(* CODESYS project Untitled1.project
   Version: 0.0.0.0
   Title: Untitled1
   Author: madsw

Project tree, tasks and I/O mapping:
  PeackPiercePredatorPendulumProtagonistINATOR_5000 : TM241CEC24T/U, Schneider Electric, order no. TM241CEC24T/U, version 5.0.8.2
      settings: OPCUA enable = True; Dummy int param for online change = 2
    application Application
      libraries: HttpHandling, 1.1.4.0 (Schneider Electric); SysMem, 3.5.12.0 (System); TcpUdpCommunication, 2.0.15.0 (Schneider Electric)
      task MAST (cyclic, interval 300 ms, priority 16, watchdog 100 ms x 1) calls SR_Main
      task MAST_1 (cyclic, interval 100 ms, priority 15, watchdog 50 ms x 1) calls POU
      task Task3 (cyclic, interval 1 ms, priority 1) calls counter
      task VISU_TASK (cyclic, interval 100 ms, priority 31) calls VisuElems.Visu_Prg
      global variables GVL
      program SR_Main [ST]
      POU - Error check functions/
        function CheckBounds [ST]
        function CheckDivDInt [ST]
        function CheckDivLInt [ST]
        function CheckDivReal [ST]
        function CheckDivLReal [ST]
        function CheckPointer [ST]
        function CheckRangeSigned [ST]
        function CheckRangeUnsigned [ST]
        function CheckLRangeSigned [ST]
        function CheckLRangeUnsigned [ST]
      program POU [ST]
      trace Trace (task ): SR_Main.do_Q0
      visualisation Visualization
      program counter [ST]
      OPCUASymbolConfiguration
    DI : Digital Inputs, Schneider Electric, version 5.0.8.2
        settings: IOs Usage = 3
        input  iwDI_IW0 : WORD  // IW0
        input  ibDI_IB1 : BYTE  // IB1
    DQ : Digital Outputs, Schneider Electric, version 5.0.8.2
        output Application.POU.lightArray[0] : BOOL  // QW0.Q0
        output Application.POU.lightArray[1] : BOOL  // QW0.Q1
        output Application.POU.lightArray[2] : BOOL  // QW0.Q2
        output Application.POU.lightArray[3] : BOOL  // QW0.Q3
        output Application.POU.lightArray[4] : BOOL  // QW0.Q4
        output Application.POU.lightArray[5] : BOOL  // QW0.Q5
        output Application.POU.lightArray[6] : BOOL  // QW0.Q6
        output Application.POU.lightArray[7] : BOOL  // QW0.Q7
        output Application.POU.lightArray[8] : BOOL  // QW0.Q8
        output Application.POU.lightArray[9] : BOOL  // QW0.Q9
        output qbDQ_QB1 : BYTE  // QB1
        unmapped channels: QW0
    Counters : Counters, Schneider Electric, version 5.0.8.2
        settings: Instance name = 'HscMainDualPhase_0'; B input History = 'old=-1 new=1'; A input History = 'old=-1 new=0'; Temporary Instance name = 'HscMainDualPhase_0'
    Pulse_Generators : Pulse Generators, Schneider Electric, version 5.0.8.2
    Cartridge_1 : Cartridge, Schneider Electric, version 5.0.8.2
    IO_Bus : IO bus - TM3, Schneider Electric, version 5.0.8.2
      Module_1 : TM3SAF5R/G, Schneider Electric, order no. TM3SAF5R/G, version 1.0.1.14
          input  iwModule_1_IW0 : WORD  // IW0
          output qbModule_1_QB0 : BYTE  // QB0
      Module_2 : TM3AQ4/G, Schneider Electric, order no. TM3AQ4/G, version 1.0.0.15
          output qiModule_2_QW0 : INT  // QW0
          output qiModule_2_QW1 : INT  // QW1
          output qiModule_2_QW2 : INT  // QW2
          output qiModule_2_QW3 : INT  // QW3
          input  ibModule_2_IBStatusQW0 : BYTE  // IBStatusQW0
          input  ibModule_2_IBStatusQW1 : BYTE  // IBStatusQW1
          input  ibModule_2_IBStatusQW2 : BYTE  // IBStatusQW2
          input  ibModule_2_IBStatusQW3 : BYTE  // IBStatusQW3
    COM_Bus : COM bus, Schneider Electric, version 5.0.8.2
    Ethernet_1 : Ethernet Network, Schneider Electric, version 5.0.8.2
        settings: IPAddress = [192, 168, 0, 50]; SubnetMask = [255, 255, 255, 0]; WebServer = TRUE; FTP Server = FALSE; SoMachine Protocol = TRUE; Modbus Server = FALSE; NetManage Protocol = TRUE; SNMP protocol = FALSE; Enable Routing = FALSE; WebVisu protocol = TRUE; DHCP Server Active = TRUE
    Serial_Line_1 : Serial line, Schneider Electric, version 5.0.8.2
      Machine_Expert_Network_Manager : Machine Expert-Network Manager, Schneider Electric, version 4.0.0.3
    Serial_Line_2 : Serial line, Schneider Electric, version 5.0.8.2
      Modbus_Manager : Modbus Manager, Schneider Electric, version 4.0.0.3
    CAN_1 : CANopen bus, Schneider Electric, version 5.0.8.2
  FdtConnections : FDT Connections, Schneider Electric, version 1.0.0.2
  libraries: VisuSymbols, 3.5.10.0 (System)
  CNC settings
  text list GlobalTextList
*)

// PeackPiercePredatorPendulumProtagonistINATOR_5000/Application/GVL
{attribute 'qualified_only'}
VAR_GLOBAL
	gLightArray: ARRAY[0..8] OF BOOL;
	count: UINT;
	
	// OPC UA varibels for interface.
	G_angle: UINT := 45;
END_VAR

// PeackPiercePredatorPendulumProtagonistINATOR_5000/Application/SR_Main
PROGRAM SR_Main
// Comment
VAR
	di_I0: BOOL;
	count: UINT := 4;
	do_Q0: BOOL;
	TCPClient: TCPUDP.FB_TCPClient;
	TCPServer: TCPUDP.FB_TCPServer;
	readBuffer: BYTE;
	PID: PID;
	PD: PD;
END_VAR;

// Global light
GVL.gLightArray[count] := FALSE;
IF count >= 8 THEN
	count := 0;
ELSE
	count := count +1;	
END_IF;
GVL.gLightArray[count] := TRUE;

do_Q0 := NOT NOT NOT di_I0;


HscMainDualPhase_0.CurrentValue;
// TCPClient.Receive(ADR(readBuffer), SIZEOF(BYTE), );

END_PROGRAM

// PeackPiercePredatorPendulumProtagonistINATOR_5000/Application/POU
PROGRAM POU
VAR
	lightArray: ARRAY[0..9] OF BOOL;
	count: UINT;
END_VAR

lightArray[count] := FALSE;
GVL.gLightArray[count] := FALSE;

IF count+1 = SIZEOF(lightArray)/SIZEOF(BOOL) THEN
	count := 0;
ELSE
	count := count +1;	
END_IF;

lightArray[count] := TRUE;
GVL.gLightArray[count] := TRUE;

END_PROGRAM

// PeackPiercePredatorPendulumProtagonistINATOR_5000/Application/counter
PROGRAM counter
VAR
	ctu: CTUD;
	adasd: CTUD;
END_VAR

END_PROGRAM

// PeackPiercePredatorPendulumProtagonistINATOR_5000/Application/POU - Error check functions/CheckBounds
// Implicitly generated code : DO NOT EDIT
FUNCTION CheckBounds : DINT
VAR_INPUT
	index, lower, upper: DINT;
END_VAR

// Implicitly generated code : Only an Implementation suggestion
IF  index < lower THEN
	CheckBounds := lower;
ELSIF  index > upper THEN
	CheckBounds := upper;
ELSE  
	CheckBounds := index;
END_IF

(*It is also possible to set a breakpoint, log messages or e.g. to halt on an exception:
Add CmpApp.library, SysExcept.library and SysTypes2_Itf as newest.
Declaration:
VAR
    _pApp : POINTER TO CmpApp.APPLICATION;
    _result   : SysTypes.RTS_IEC_RESULT;
END_VAR

Implementation:
_pApp := AppGetCurrent(pResult:=_result);
IF  index < lower THEN
        CheckBounds := lower;
        IF _pApp <> 0 THEN
                AppGenerateException(pApp:=_pApp, ulException:=RtsExceptions.RTSEXCPT_ARRAYBOUNDS);
        END_IF
ELSIF  index > upper THEN
        CheckBounds := upper;
        IF _pApp <> 0 THEN
                AppGenerateException(pApp:=_pApp,   ulException:=RtsExceptions.RTSEXCPT_ARRAYBOUNDS);
        END_IF
ELSE  
        CheckBounds := index;
END_IF
*)

END_FUNCTION

// PeackPiercePredatorPendulumProtagonistINATOR_5000/Application/POU - Error check functions/CheckDivDInt
// Implicitly generated code : DO NOT EDIT
FUNCTION CheckDivDInt : DINT
VAR_INPUT
	divisor:DINT;
END_VAR

// Implicitly generated code : Only an Implementation suggestion
IF divisor = 0 THEN
	CheckDivDInt:=1;
ELSE
	CheckDivDInt:=divisor;
END_IF;

END_FUNCTION

// PeackPiercePredatorPendulumProtagonistINATOR_5000/Application/POU - Error check functions/CheckDivLInt
// Implicitly generated code : DO NOT EDIT
FUNCTION CheckDivLInt : LINT
VAR_INPUT
	divisor:LINT;
END_VAR

// Implicitly generated code : Only an Implementation suggestion
IF divisor = 0 THEN
	CheckDivLInt:=1;
ELSE
	CheckDivLInt:=divisor;
END_IF;

END_FUNCTION

// PeackPiercePredatorPendulumProtagonistINATOR_5000/Application/POU - Error check functions/CheckDivReal
// Implicitly generated code : DO NOT EDIT
FUNCTION CheckDivReal : REAL
VAR_INPUT
	divisor:REAL;
END_VAR

// Implicitly generated code : Only an Implementation suggestion
IF divisor = 0 THEN
	CheckDivReal:=1;
ELSE
	CheckDivReal:=divisor;
END_IF;

END_FUNCTION

// PeackPiercePredatorPendulumProtagonistINATOR_5000/Application/POU - Error check functions/CheckDivLReal
// Implicitly generated code : DO NOT EDIT
FUNCTION CheckDivLReal : LREAL
VAR_INPUT
	divisor:LREAL;
END_VAR

// Implicitly generated code : Only an Implementation suggestion
IF divisor = 0 THEN
	CheckDivLReal:=1;
ELSE
	CheckDivLReal:=divisor;
END_IF;

END_FUNCTION

// PeackPiercePredatorPendulumProtagonistINATOR_5000/Application/POU - Error check functions/CheckPointer
// Implicitly generated code : DO NOT EDIT
FUNCTION CheckPointer : POINTER TO BYTE
VAR_INPUT 
	ptToTest : POINTER TO BYTE; // Destination address of the pointer
	iSize : DINT;		        // Size of the type the pointer points to. (e.g: 20 for POINTER TO ARRAY [0..9] OF INT) 
	iGran : DINT;		        // Granularity of the pointer access. This is the size of the biggest non-structured data type in the type the pointer points to. (e.g: 2 for POINTER TO ARRAY [0..9] OF INT)
	bWrite: BOOL;		        // Indicates read or write Access. TRUE = write access.
END_VAR

// No standard way of implementation. Fill your own code here
CheckPointer := ptToTest;

END_FUNCTION

// PeackPiercePredatorPendulumProtagonistINATOR_5000/Application/POU - Error check functions/CheckRangeSigned
// Implicitly generated code : DO NOT EDIT
FUNCTION CheckRangeSigned : DINT
VAR_INPUT
	value, lower, upper: DINT;
END_VAR

// Implicitly generated code : Only an Implementation suggestion
IF (value < lower) THEN
	CheckRangeSigned := lower;
ELSIF(value > upper) THEN
	CheckRangeSigned := upper;
ELSE
	CheckRangeSigned := value;
END_IF

END_FUNCTION

// PeackPiercePredatorPendulumProtagonistINATOR_5000/Application/POU - Error check functions/CheckRangeUnsigned
// Implicitly generated code : DO NOT EDIT
FUNCTION CheckRangeUnsigned : UDINT
VAR_INPUT
	value, lower, upper: UDINT;
END_VAR

// Implicitly generated code : Only an Implementation suggestion
IF (value < lower) THEN
	CheckRangeUnsigned := lower;
ELSIF(value > upper) THEN
	CheckRangeUnsigned := upper;
ELSE
	CheckRangeUnsigned := value;
END_IF

END_FUNCTION

// PeackPiercePredatorPendulumProtagonistINATOR_5000/Application/POU - Error check functions/CheckLRangeSigned
// Implicitly generated code : DO NOT EDIT
FUNCTION CheckLRangeSigned : LINT
VAR_INPUT
	value, lower, upper: LINT;
END_VAR

// Implicitly generated code : Only an Implementation suggestion
IF (value < lower) THEN
	CheckLRangeSigned := lower;
ELSIF(value > upper) THEN
	CheckLRangeSigned := upper;
ELSE
	CheckLRangeSigned := value;
END_IF

END_FUNCTION

// PeackPiercePredatorPendulumProtagonistINATOR_5000/Application/POU - Error check functions/CheckLRangeUnsigned
// Implicitly generated code : DO NOT EDIT
FUNCTION CheckLRangeUnsigned : ULINT
VAR_INPUT
	value, lower, upper: ULINT;
END_VAR

// Implicitly generated code : Only an Implementation suggestion
IF (value < lower) THEN
	CheckLRangeUnsigned := lower;
ELSIF(value > upper) THEN
	CheckLRangeUnsigned := upper;
ELSE
	CheckLRangeUnsigned := value;
END_IF

END_FUNCTION

// PeackPiercePredatorPendulumProtagonistINATOR_5000/Application/Visualization
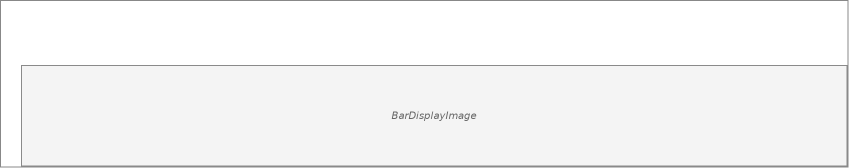
VISUALIZATION Visualization  // 849x168
    BarDisplayImage (21,65 826x101), value: GVL.G_angle, style: BarDisplayImage-Gray, scale format: %.1f, scale 0..360
END_VISUALIZATION
